FUNCTION_BLOCK PVFORECASTER_DEB (* Function block for holding historical PV power measurements and generating PV power forecasts. *)
  (* Standard: 61499-2; Description: IEC 61499 implementation of the "PVprog" algorithm. Original version's MIT license: Copyright (c) 2016 Joseph Bergner, Johannes Weniger, Tjarko Tjaden Permission is hereby granted, free of charge, to any person obtaining a copy of this software and associated documentation files (the "Software"), to deal in the Software without restriction, including without limitation the rights to use, copy, modify, merge, publish, distribute, sublicense, and/or sell copies of the Software, and to permit persons to whom the Software is furnished to do so, subject to the following conditions: The above copyright notice and this permission notice shall be included in all copies or substantial portions of the Software. THE SOFTWARE IS PROVIDED "AS IS", WITHOUT WARRANTY OF ANY KIND, EXPRESS OR IMPLIED, INCLUDING BUT NOT LIMITED TO THE WARRANTIES OF MERCHANTABILITY, FITNESS FOR A PARTICULAR PURPOSE AND NONINFRINGEMENT. IN NO EVENT SHALL THE AUTHORS OR COPYRIGHT HOLDERS BE LIABLE FOR ANY CLAIM, DAMAGES OR OTHER LIABILITY, WHETHER IN AN ACTION OF CONTRACT, TORT OR OTHERWISE, ARISING FROM, OUT OF OR IN CONNECTION WITH THE SOFTWARE OR THE USE OR OTHER DEALINGS IN THE SOFTWARE. *)
  (* Version 0.0, 2017-05-03, 4DIAC-IDE, 4DIAC-Consortium *)
  (* Version 1.0, 2017-05-03, Marc Jakobi, HTW Berlin *)
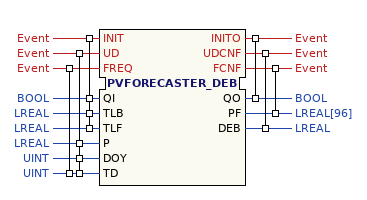
  EVENT_INPUT
    INIT WITH QI, TLB, TLF; (* Initialization Request *)
    UD WITH P, TD, DOY; (* PV Forecast Update Request *)
    FREQ WITH TD; (* Forecast Request *)
  END_EVENT
  EVENT_OUTPUT
    INITO WITH QO; (* Initialization Confirm *)
    UDCNF WITH DEB; (* Update Algorithm Execution Confirmation *)
    FCNF WITH PF; (* Forecast Confirmation *)
  END_EVENT
  VAR_INPUT
    QI : BOOL; (* Input event qualifier *)
    TLB : LREAL := 3; (* Time frame to look back when generating forecasts in h *)
    TLF : LREAL := 15; (* Time frame to forecast ahead (look forward) in h *)
    P : LREAL; (* Measured PV power in W *)
    DOY : UINT := 1; (* Day of the year [1..365] *)
    TD : UINT := 0; (* Time of day [min] [0..1439] *)
  END_VAR
  VAR_OUTPUT
    QO : BOOL; (* Output event qualifier *)
    PF : ARRAY [0..95] OF LREAL; (* Forecasted PV power *)
    DEB : LREAL; (* Debug output *)
  END_VAR
  VAR
    PVMAXLASTDAY : ARRAY [0..1439] OF LREAL; (* Maximum PV power over last 10 days (approximation of what the PV power would be on a clear sky day) [W]. Used for generating the PV forecast. *)
    PVMAXBEFORELASTDAY : ARRAY [0..1439] OF LREAL; (* Maximum PV power over last 10 days (1 day before PVMAXLASTDAY) [W] *)
    PVMAXCURRDAY : ARRAY [0..1439] OF LREAL; (* Maximum PV power over last 10 days (used for generating PVMAXLASTDAY) [W] *)
    PVMAX15LASTDAY : ARRAY [0..95] OF LREAL; (* 15 min average of PVMAXLASTDAY [W] *)
    PVMAX15CURRDAY : ARRAY [0..95] OF LREAL; (* 15 min average of PVMAXCURRDAY [W] *)
    LASTMAX : ARRAY [0..14399] OF LREAL; (* Cache used to recalculate PVMAXCURRDAY if the last maximum is more than 10 days old [W] *)
    LASTMAXAGE : ARRAY [0..1439] OF UINT; (* Stores the age [d] of the last calculated PV power PVMAXCURRDAY for each [time of day] to reduce recalculation of PVMAXCURRDAY *)
    AGEINDEX : UINT := 1; (* Index used for storing LASTMAX according to its age (see LASTMAXAGE). Increments between 1 and 1440 every minute and resets after reaching 1440. *)
    ENERGYCLEARNESSINDEX : ARRAY [0..1439] OF LREAL; (* Forecasted Clearness Index of the PV energy (equivalent to the fraction of the actual energy and the energy without clouds) *)
    LOOKBACKTIMEINTIMESTEPS : UINT; (* Number of time steps (minutes) to look back when generating forecasts *)
    LOOKFORWARDTIMEINTIMESTEPS : UINT; (* Number of time steps (15 min intervals) to look ahead for forecast *)
    LOOKBACKTIMEINHOURS : LREAL; (* Time frame to look back when generating forecasts in h *)
    LOOKFORWARDTIMEINHOURS : LREAL; (* Time frame to forecast ahead in h *)
    POWERLASTDAY : ARRAY [0..1439] OF LREAL; (* Stores the historical PV power [W] of the last day *)
    POWERCURRDAY : ARRAY [0..1439] OF LREAL; (* Stores the historical PV power [W] of the current day *)
    LASTTIMESTEP : INT := -1; (* Time at the point of the last call of the prepareForecast algorithm *)
    LASTDAYOFYEAR : UINT := 0; (* Day of the year [1...365] of the last call of the prepareForecast algorithm *)
    TIMESINCELASTUPDATE : INT := 1; (* Time [min] between last update and current one *)
    LASTMEASUREDPOWER : LREAL := 0; (* Power P [W] input when last update occurred *)
    PU : LREAL := 0; (* Power (either current or interpolated) [W] used for updating memory *)
    TIMEINDEX : UINT := 0; (* Time index (either current or interpolated) [min] used for updating memory *)
  END_VAR
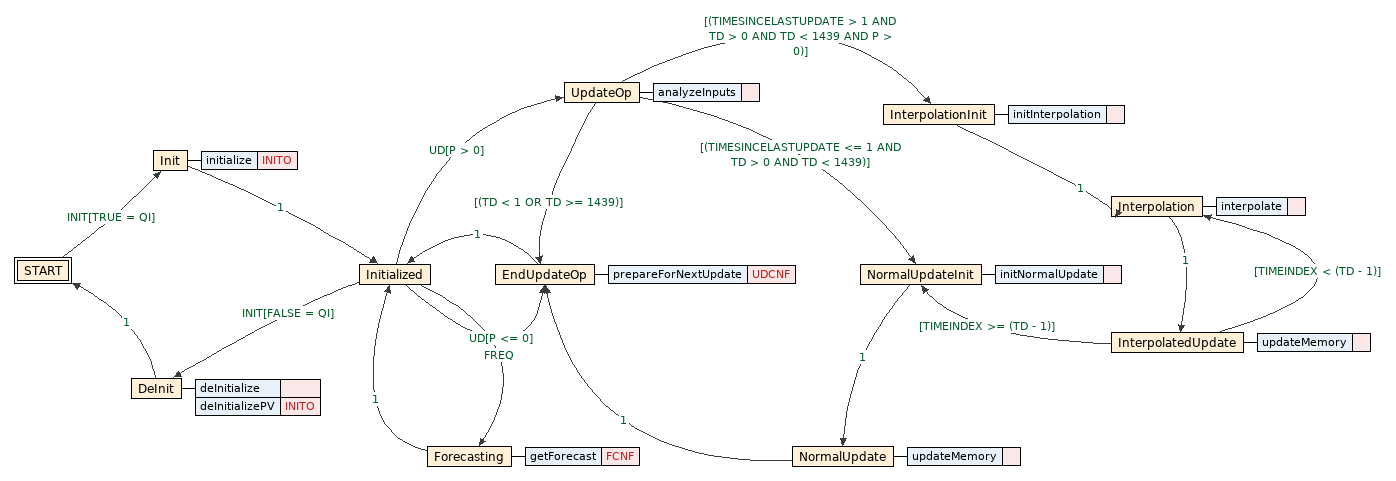
  EC_STATES
    START; (* Initial State *)
    Init : initialize -> INITO; (* Initialization *)
    UpdateOp : analyzeInputs; (* Normal execution *)
    Initialized;
    DeInit : deInitialize, deInitializePV -> INITO;
    Forecasting : getForecast -> FCNF;
    Interpolation : interpolate;
    NormalUpdate : updateMemory;
    EndUpdateOp : prepareForNextUpdate -> UDCNF;
    InterpolatedUpdate : updateMemory;
    NormalUpdateInit : initNormalUpdate;
    InterpolationInit : initInterpolation;
  END_STATES
  EC_TRANSITIONS
    DeInit TO START := 1;
    START TO Init := INIT[TRUE = QI];
    Init TO Initialized := 1;
    Initialized TO DeInit := INIT[FALSE = QI];
    Forecasting TO Initialized := 1;
    Initialized TO Forecasting := FREQ;
    EndUpdateOp TO Initialized := 1;
    UpdateOp TO EndUpdateOp := [(TD < 1 OR TD >= 1439)];
    NormalUpdate TO EndUpdateOp := 1;
    UpdateOp TO NormalUpdateInit := [(TIMESINCELASTUPDATE <= 1 AND TD > 0 AND TD < 1439)];
    UpdateOp TO InterpolationInit := [(TIMESINCELASTUPDATE > 1 AND TD > 0 AND TD < 1439 AND P > 0)];
    InterpolationInit TO Interpolation := 1;
    Interpolation TO InterpolatedUpdate := 1;
    InterpolatedUpdate TO Interpolation := [TIMEINDEX < (TD - 1)];
    InterpolatedUpdate TO NormalUpdateInit := [TIMEINDEX >= (TD - 1)];
    NormalUpdateInit TO NormalUpdate := 1;
    Initialized TO UpdateOp := UD[P > 0];
    Initialized TO EndUpdateOp := UD[P <= 0];
  END_TRANSITIONS
  ALGORITHM initialize IN ST: (* Initialization algorithm *)
VAR
	tmp1 : LREAL;
	tmp2 : UINT;
END_VAR;
/*
 * Used internal vars & inputs:
 * TLB, TLF, LOOKBACKTIMEINHOURS, LOOKFORWARDTIMEINHOURS : LREAL;
 * LOOKBACKTIMEINTIMESTEPS, LOOKFORWARDTIMEINTIMESTEPS : UINT;
 * QO : BOOL;
 */
// Limit inputs to acceptable boundaries
IF TLB < 0 THEN
	TLB := 0;
ELSIF TLB > 24 THEN
	TLB := 24;
END_IF;
LOOKBACKTIMEINHOURS := TLB;
// Workaround for ceil function
tmp1 := LOOKBACKTIMEINHOURS * 60; // input resolution = 1 min
tmp2 := LREAL_TO_UINT(tmp1);
IF UINT_TO_LREAL(tmp2) < tmp1 THEN
 	LOOKBACKTIMEINTIMESTEPS := tmp2 + 1;
ELSE
	LOOKBACKTIMEINTIMESTEPS := tmp2;
END_IF;
// Set forecast horizon
IF TLF < 0 THEN
	TLF := 0;
ELSIF TLF > 24 THEN
	TLF := 24;
END_IF;
LOOKFORWARDTIMEINHOURS := TLF;
tmp1 := LOOKFORWARDTIMEINHOURS * 4; // output resolution = 15 min
tmp2 := LREAL_TO_UINT(tmp1);
IF UINT_TO_LREAL(tmp2) < tmp1 THEN
 	LOOKFORWARDTIMEINTIMESTEPS := tmp2 + 1;
ELSE
	LOOKFORWARDTIMEINTIMESTEPS := tmp2;
END_IF;
QO := QI; // Pass Input event qualifier to output event qualifier
  END_ALGORITHM
  ALGORITHM deInitialize IN ST: (* Deinitialization algorithm *)
VAR
	j : UINT;
END_VAR;
/*
 * Used internal vars & inputs:
 * POWERCURRDAY, POWERLASTDAY, LASTMEASUREDPOWER : LREAL;
 * LASTDAYOFYEAR : UINT;
 * LASTTIMESTEP : INT;
 * QO : BOOL;
 */
// Reset all internal variables to initial values
FOR j := 0 TO 1439 BY 1 DO
	POWERCURRDAY[j] := 0;
	POWERLASTDAY[j] := 0;
END_FOR;
LASTDAYOFYEAR := 0;
LASTTIMESTEP := -1;
LASTMEASUREDPOWER := 0;
QO := FALSE;
  END_ALGORITHM
  ALGORITHM analyzeInputs IN ST: (* Stores PV data and prepares it for forecast generation *)
VAR
	i : UINT;
END_VAR;
/*
 * Used internal vars & inputs:
 * AGEINDEX, DOY, LASTDAYPFYEAR, TD : UINT;
 * TIMESINCELASTUPDATE, LASTTIMESTEP : INT;
 * POWERLASTDAY, POWERCURRDAY, PVMAXBEFORELASTDAY, PVMAXLASTDAY, PVMAXLASTDAY, PVMAX15LASTDAY, PVMAX15CURRDAY : LREAL;
 */
TIMESINCELASTUPDATE := UINT_TO_INT(TD) - LASTTIMESTEP;
// At the beginning of each day, replace LASTDAY arrays with CURRDAY arrays
IF DOY <> LASTDAYOFYEAR THEN
	FOR i := 0 TO 1439 BY 1 DO
		POWERLASTDAY[i] := POWERCURRDAY[i];
		PVMAXBEFORELASTDAY[i] := PVMAXLASTDAY[i];
		PVMAXLASTDAY[i] := PVMAXCURRDAY[i];
	END_FOR;
	FOR i := 0 TO 95 BY 1 DO
		PVMAX15LASTDAY[i] := PVMAX15CURRDAY[i];
	END_FOR;
	LASTDAYOFYEAR := DOY;
	// Increment AGEINDEX and reset at 10
	AGEINDEX := AGEINDEX + 1;
	IF AGEINDEX > 10 THEN
		AGEINDEX := 1;
	END_IF;
	TIMESINCELASTUPDATE := 1; // Set to 1 minute for beginning of day
END_IF;
  END_ALGORITHM
  ALGORITHM getForecast IN ST: (* Generates forecast from currently stored PV data *)
VAR
	td15 : UINT;
	j : INT;
	ind : INT;
	switchdoy : BOOL;
	tmpI : INT;
	meanClearnessIndex : LREAL;
END_VAR;
/*
 * Used internal vars & inputs:
 * DOY, TD, LOOKFORWARDTIMEINTIMESTEPS : UINT;
 * PF, PVMAX15CURRDAY, PVMAX15LASTDAY : LREAL;
 */
td15 := TD / 15; // Time of day in 15 min intervals
meanClearnessIndex := ENERGYCLEARNESSINDEX[TD]; // 15 min mean of ENERGYCLEARNESSINDEX (kT)
// Calculate 15 minute mean of PVMAXCURRDAY and ENERGYCLEARNESSINDEX
PVMAX15CURRDAY[td15] := PVMAXCURRDAY[TD];
// tmpI := MAX(0, TD - 14);
tmpI := UINT_TO_INT(TD) -  14; // Temporary variable for setting loop index's lower limit to 0
IF tmpI < 0 THEN
	tmpI := 0;
END_IF;
FOR j := tmpI TO UINT_TO_INT(TD) - 1 BY 1 DO
	meanClearnessIndex := meanClearnessIndex + ENERGYCLEARNESSINDEX[j];
	PVMAX15CURRDAY[td15] := PVMAX15CURRDAY[td15] + PVMAXCURRDAY[j];
END_FOR;
IF meanClearnessIndex > 0 THEN
	meanClearnessIndex := meanClearnessIndex / 15;
ELSE // Set night time clearnessIndex to 1 so that PV power forecasts appear before the end of the night (better for load peak shaving)
	meanClearnessIndex := 1;
END_IF;
IF PVMAX15CURRDAY[td15] > 0 THEN
	PVMAX15CURRDAY[td15] := PVMAX15CURRDAY[td15] / 15;
END_IF;
// Iterate through PVMAX15LASTDAY and multiply each element with KTF15 to generate PV forecast
ind := td15;  // Index variable to determine if day caches must be switched
switchdoy := FALSE; // Flag for switching day caches
FOR j := td15 TO td15 + LOOKFORWARDTIMEINTIMESTEPS - 1 BY 1 DO
	IF ind >= 96 THEN
		ind := 0;
		switchdoy := TRUE;
	END_IF;
	IF switchdoy THEN
		PF[j - td15] := meanClearnessIndex * PVMAX15CURRDAY[ind];
	ELSE
		PF[j - td15] := meanClearnessIndex * PVMAX15LASTDAY[ind];
	END_IF;
	ind := ind + 1;
END_FOR;
  END_ALGORITHM
  ALGORITHM updateMemory IN ST: (* Updates the memory with measured or interpolated PV data *)
VAR
	pvMax : LREAL;
	pastPVenergy : LREAL;
	maxPVenergy : LREAL;
	incrementAge : BOOL;
	switchDays : BOOL;
	j : UINT;
	timeStepCounter : UINT;
	switchDayCounter : UINT;
	ind: INT;
END_VAR;
/*
 * Used internal vars & inputs:
 * PU, POWERCURRDAY, POWERLASTDAY, PVMAXLASTDAY PVMAXBEFORELASTDAY, LASTMAX, ENERGYCLEARNESSINDEX  : LREAL;
 * TIMEINDEX, LASTMAXAGE, AGEINDEX  : UINT;
 */
// Initialize local variables
timeStepCounter := 0; // counter for ENERGYCLEARNESSINDEX (kT) calculation
switchDays := FALSE; // Flag to indicate switching between CurrDay and LastDay for kT calculation
switchDayCounter := 0; // counter for kT calculation
pastPVenergy := 0; // kT := MIN(1, pastPVenergy / maxPVenergy);
// Save current power measurement
POWERCURRDAY[TIMEINDEX + 1] := PU;
// Update cache
LASTMAX[(AGEINDEX - 1) * 1440 + TIMEINDEX] := PU; // converted 2D array index to 1D array index due to 4diac lacking support for 2D arrays
pvMax := PVMAXLASTDAY[TIMEINDEX]; // maximum PV power of last 10 days at TIMEINDEX
IF PU > pvMax THEN // workaround for MAX() function
 	pvMax := PU;
END_IF;
incrementAge := TRUE; // Remains TRUE if AGEINDEX is to be incremented
/*
 * Iterate through values at same time of day of the cached last 10 days to find a new maximum value
 * if the current maximum value is 10 days old i.e. if no new maximum turns up for longer than 10 days.
 */
IF LASTMAXAGE[TIMEINDEX] >= 9 THEN
	pvMax := PU;
	FOR j := AGEINDEX TO 1 BY -1 DO
		IF LASTMAX[(j - 1) * 1440 + TIMEINDEX] > pvMax THEN
			LASTMAXAGE[TIMEINDEX] := AGEINDEX - j; // calculate age of next pvMax
			pvMax := LASTMAX[(j - 1) * 1440 + TIMEINDEX]; // set pvMax to found last maximum that is less than 10 days old
			incrementAge := FALSE;
		END_IF;
	END_FOR;
	FOR j := 10 TO AGEINDEX + 1 BY -1 DO
		IF LASTMAX[(j - 1) * 1440 + TIMEINDEX] > pvMax THEN
			LASTMAXAGE[TIMEINDEX] := 10 - j + AGEINDEX; // calculate age of next pvMax
			pvMax := LASTMAX[(j - 1) * 1440 + TIMEINDEX];
			incrementAge := FALSE;
		END_IF;
	END_FOR;
END_IF;
IF PU = pvMax THEN
	LASTMAXAGE[TIMEINDEX] := 0; // Reset age if current power greater than last max
ELSIF PU < pvMax AND incrementAge THEN // Otherwise increment age if no new maximum was found in LASTMAX and old maximum was older than 10 days
	LASTMAXAGE[TIMEINDEX] := LASTMAXAGE[TIMEINDEX] + 1;
END_IF;
PVMAXCURRDAY[TIMEINDEX] := pvMax; // save pvMax
// Calculate ENERGYCLEARNESSINDEX
ind := UINT_TO_INT(TIMEINDEX);
WHILE timeStepCounter < LOOKBACKTIMEINTIMESTEPS AND switchDayCounter < 2 DO
	// Reset j to end of day and switch to LastDay if j reaches zero
	IF ind < 0 THEN
		ind := 1439;
		switchDays := TRUE;
		switchDayCounter := switchDayCounter + 1;
	END_IF;
	// Only add daytime values
	IF (switchDays AND POWERLASTDAY[ind] > 0) THEN
		pastPVenergy := pastPVenergy + POWERLASTDAY[ind];
		maxPVenergy := maxPVenergy + PVMAXBEFORELASTDAY[ind];
		timeStepCounter := timeStepCounter + 1;
	ELSIF (NOT switchDays) AND POWERCURRDAY[ind] > 0 THEN
			pastPVenergy := pastPVenergy + POWERCURRDAY[ind];
			maxPVenergy := maxPVenergy + PVMAXLASTDAY[ind];
			timeStepCounter := timeStepCounter + 1;
	END_IF;
	IF PU = 0 THEN
		pastPVenergy := 0;
		maxPVenergy := 0;
	END_IF;
	ind := ind - 1;
END_WHILE;
IF (pastPVenergy = 0 OR maxPVenergy = 0 OR PU = 0) THEN // Set to 1 at night time or when division by 0 would occur
	ENERGYCLEARNESSINDEX[TIMEINDEX + 1] := 1;
ELSE
	ENERGYCLEARNESSINDEX[TIMEINDEX + 1] := pastPVenergy / maxPVenergy;
	IF ENERGYCLEARNESSINDEX[TIMEINDEX + 1] > 1 THEN // kT cannot be greater than 1
		ENERGYCLEARNESSINDEX[TIMEINDEX + 1] := 1;
	END_IF;
END_IF;
  END_ALGORITHM
  ALGORITHM interpolate IN ST: (* Interpolates between last and currently measured PV data *)
/*
 * Used internal vars & inputs:
 * INTERPOLATIONINCREMENT, LASTMEASUREDPOWER, P, PU  : LREAL;
 * TD, TIMEINDEX  : UINT;
 */
// Linear interpolation between last measured power and currently measured power
PU := PU + (P - LASTMEASUREDPOWER) / INT_TO_LREAL(TIMESINCELASTUPDATE);
TIMEINDEX := TIMEINDEX + 1;
  END_ALGORITHM
  ALGORITHM prepareForNextUpdate IN ST: (* Saves the current inputs for next update *)
/*
 * Used internal vars & inputs:
 * LASTMEASUREDPOWER : LREAL;
 * LASTTIMESTEP : INT;
 * TD : UINT;
 */
LASTMEASUREDPOWER := P;
LASTTIMESTEP := UINT_TO_INT(TD);
  END_ALGORITHM
  ALGORITHM initNormalUpdate IN ST: (* Sets memory update inputs PU and TIMEINDEX to current values *)
/*
 * Used internal vars & inputs:
 * P, PU : LREAL;
 * TD, TIMEINDEX : UINT;
 */
PU := P;
TIMEINDEX := TD - 1; //subtract 1 from time of day for correct indexing
  END_ALGORITHM
  ALGORITHM initInterpolation IN ST: (* Sets tieme index to initialize interpolation *)
/*
 * Used internal vars & inputs:
 * TD, TIMEINDEX : UINT;
 * TIMESINCELASTUPDATE : INT;
 * LASTMEASUREDPOWER, PU : LREAL;
 */
 // Initialize TIMEINDEX and PU for interpolation
TIMEINDEX := TD - INT_TO_UINT(TIMESINCELASTUPDATE);
PU := LASTMEASUREDPOWER;
  END_ALGORITHM
  ALGORITHM deInitializePV IN ST: (* PVForecaster-specific deinitialization *)
// PVForecaster-specific de-initialization algorithm
VAR
	j : UINT;
END_VAR;
/*
 * Used internal vars & inputs:
 * PVMAXCURRDAY, PVMAXLASTDAY, PVMAXBEFORELASTDAY, ENERGYCLEARNESSINDEX,  PVMAX15LASTDAY, PVMAX15CURRDAY, LASTMAX : LREAL;
 * AGEINDEX, : UINT;
 */
// Reset all internal variables to initial values
FOR j := 0 TO 1439 BY 1 DO
	PVMAXCURRDAY[j] := 0;
	PVMAXLASTDAY[j] := 0;
	PVMAXBEFORELASTDAY[j] := 0;
	LASTMAXAGE[j] := 0;
	ENERGYCLEARNESSINDEX[j] := 0;
END_FOR;
FOR j := 0 TO 14399 BY 1 DO
	LASTMAX[j] := 0;
END_FOR;
FOR j := 0 TO 95 BY 1 DO
	PVMAX15LASTDAY[j] := 0;
	PVMAX15CURRDAY[j] := 0;
END_FOR;
AGEINDEX := 1;
  END_ALGORITHM
END_FUNCTION_BLOCK
